// TwinCAT 3 PLC project PLC
// ProgramVersion: 3.1.4024.0
// libraries:
//   Tc2_MC2, * (Beckhoff Automation GmbH)
//   Tc2_Standard, * (Beckhoff Automation GmbH)
//   Tc2_System, * (Beckhoff Automation GmbH)
//   Tc3_Module, * (Beckhoff Automation GmbH)
// project tree:
//   GVLs/ GVL.TcGVL
//   / PlcTask.TcTTO
//   POUs/ MAIN.TcPOU
// real-time tasks:
//   TASK PlcTask: cycle T#10ms, priority 20, ADS port 350
// motion (NC):
//   TASK NC-Task 1 SAF: cycle T#2ms, priority 4, ADS port 501
//   TASK NC-Task 1 SVB: cycle T#10ms, priority 8, ADS port 511
//   AXIS Asse 1 (id 1)
//     OtherSettings: AllowMotionCmdToSlave=true
//     encoder EncType=1
//     drive DrvType=5
//       Analog: TorqueSetpointScale=10, ScaleFactorActTorque=0.1
//       TimeComp: TaskDelayCycles=1
//     controller CtrType=1
//       CtrPara: PriorControlFactor=1
//         Observer: BandWidth=20
// variable links:
//   PLC/PLC Instance <-> NC-Task 1 SAF/Axes/Asse 1
//     PlcTask Inputs/GVL.axis.NcToPlc <-> Outputs/ToPlc
//     PlcTask Outputs/GVL.axis.PlcToNc <-> Inputs/FromPlc

CONFIGURATION PLC
    RESOURCE PLC ON TwinCAT3
        TASK PlcTask(INTERVAL := T#10ms, PRIORITY := 20);
        PROGRAM MAIN WITH PlcTask : MAIN;
    END_RESOURCE
END_CONFIGURATION

// ---- GVLs/GVL.TcGVL
{attribute 'qualified_only'}
VAR_GLOBAL
	//Input
	bUltrasonicSensor: BOOL;
	bUpperLimitSwitch: BOOL;
	bLowerLimitSwitch: BOOL;
	bPhotocell: BOOL;
	
	//Output
	nMotorPosition: REAL;
	bMotorUp: BOOL;
	bMotorDown: BOOL;
	
	//Internal
	axis: AXIS_REF;
	bTimeExpired: BOOL;
	fBJog: MC_Jog;
	fBPower: MC_Power;
	fBTon: TON;
END_VAR

// ---- POUs/MAIN.TcPOU
PROGRAM MAIN
VAR
END_VAR

RilevamentoVeicolo();
MovimentazionePorta();
GestioneChiusura();

ACTION GestioneChiusura:
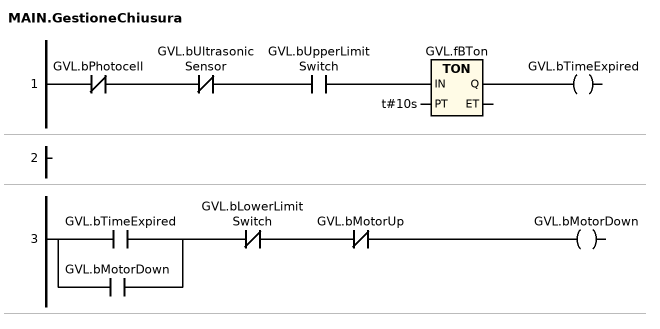
// NETWORK 1
GVL.fBTon(IN := NOT GVL.bPhotocell AND NOT GVL.bUltrasonicSensor AND GVL.bUpperLimitSwitch, PT := t#10s); // TON
GVL.bTimeExpired := GVL.fBTon.Q;

// NETWORK 2

// NETWORK 3
GVL.bMotorDown := (GVL.bTimeExpired OR GVL.bMotorDown) AND NOT GVL.bLowerLimitSwitch AND NOT GVL.bMotorUp;
END_ACTION

ACTION MovimentazionePorta:
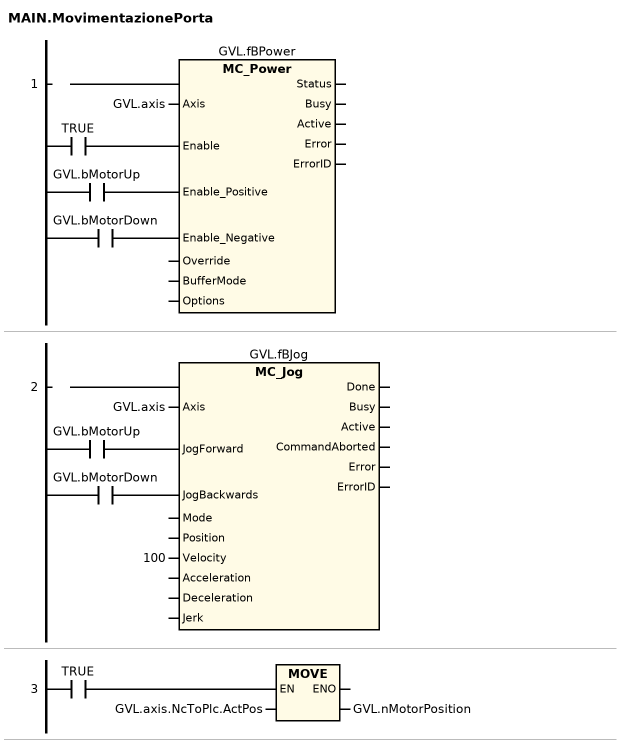
// NETWORK 1
GVL.fBPower(
    Axis := GVL.axis,
    Enable := TRUE,
    Enable_Positive := GVL.bMotorUp,
    Enable_Negative := GVL.bMotorDown); // MC_Power

// NETWORK 2
GVL.fBJog(Axis := GVL.axis, JogForward := GVL.bMotorUp, JogBackwards := GVL.bMotorDown, Velocity := 100); // MC_Jog

// NETWORK 3
GVL.nMotorPosition := GVL.axis.NcToPlc.ActPos;
END_ACTION

ACTION RilevamentoVeicolo:
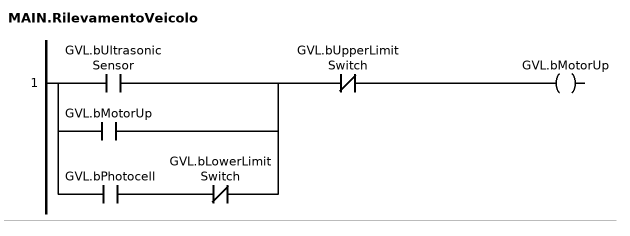
// NETWORK 1
GVL.bMotorUp := (GVL.bUltrasonicSensor OR GVL.bMotorUp OR GVL.bPhotocell AND NOT GVL.bLowerLimitSwitch) AND NOT GVL.bUpperLimitSwitch;
END_ACTION

END_PROGRAM
